% RSLogix 500 project Project_2.RSS, saved by version 8.30.00.16 %
PROJECT "UNTITLED"    % processor: Bul.1763 MicroLogix 1100 Series A %

PROGRAM FILES
  LAD 2   3 rungs
  LAD 3 "IO"  8 rungs  % Digital IO %
  LAD 4 "LOGIC"  12 rungs

DATA FILES
  O0 OUTPUT  4 elements
  I1 INPUT  6 elements
  S2 STATUS  66 elements
  B3 BINARY  1 elements
  T4 TIMER  4 elements
  C5 COUNTER  1 elements
  R6 CONTROL  1 elements
  N7 INTEGER  1 elements
  F8 FLOAT  1 elements

LADDER 2
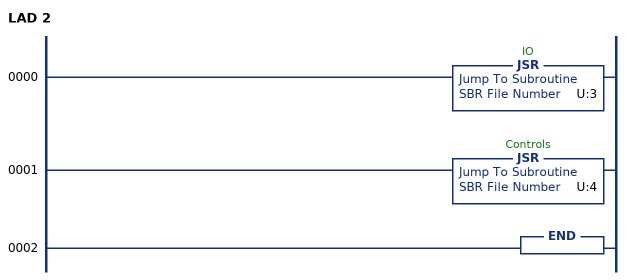
% Rung: 0 %
SOR JSR U:3 EOR
%   U:3  "IO" %
% Rung: 1 %
SOR JSR U:4 EOR
%   U:4  "Controls" %
% Rung: 2 %
SOR END EOR

LADDER 3 "IO"    % Digital IO %
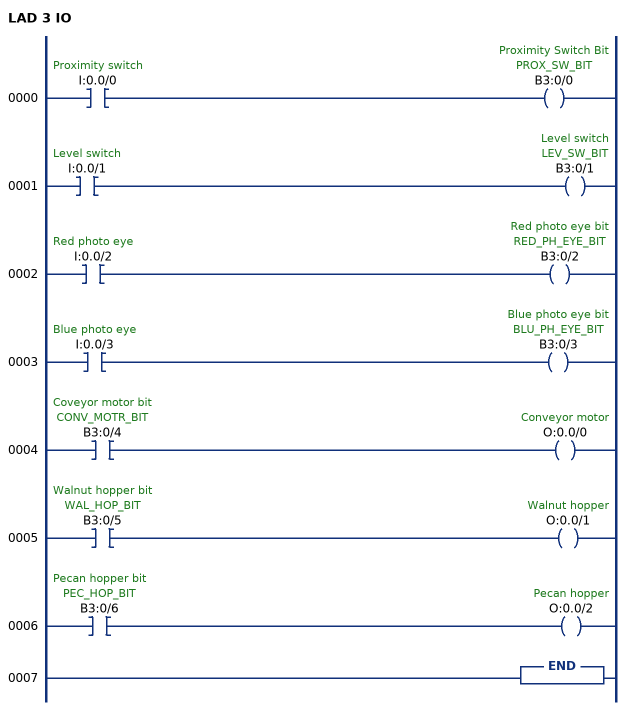
% Rung: 0 %
SOR XIC I:0.0/0 OTE B3:0/0 EOR
%   I:0.0/0  "Proximity switch" %
%   B3:0/0  PROX_SW_BIT  "Proximity Switch Bit" %
% Rung: 1 %
SOR XIC I:0.0/1 OTE B3:0/1 EOR
%   I:0.0/1  "Level switch" %
%   B3:0/1  LEV_SW_BIT  "Level switch" %
% Rung: 2 %
SOR XIC I:0.0/2 OTE B3:0/2 EOR
%   I:0.0/2  "Red photo eye" %
%   B3:0/2  RED_PH_EYE_BIT  "Red photo eye bit" %
% Rung: 3 %
SOR XIC I:0.0/3 OTE B3:0/3 EOR
%   I:0.0/3  "Blue photo eye" %
%   B3:0/3  BLU_PH_EYE_BIT  "Blue photo eye bit" %
% Rung: 4 %
SOR XIC B3:0/4 OTE O:0.0/0 EOR
%   B3:0/4  CONV_MOTR_BIT  "Coveyor motor bit" %
%   O:0.0/0  "Conveyor motor" %
% Rung: 5 %
SOR XIC B3:0/5 OTE O:0.0/1 EOR
%   B3:0/5  WAL_HOP_BIT  "Walnut hopper bit" %
%   O:0.0/1  "Walnut hopper" %
% Rung: 6 %
SOR XIC B3:0/6 OTE O:0.0/2 EOR
%   B3:0/6  PEC_HOP_BIT  "Pecan hopper bit" %
%   O:0.0/2  "Pecan hopper" %
% Rung: 7 %
SOR END EOR

LADDER 4 "LOGIC"
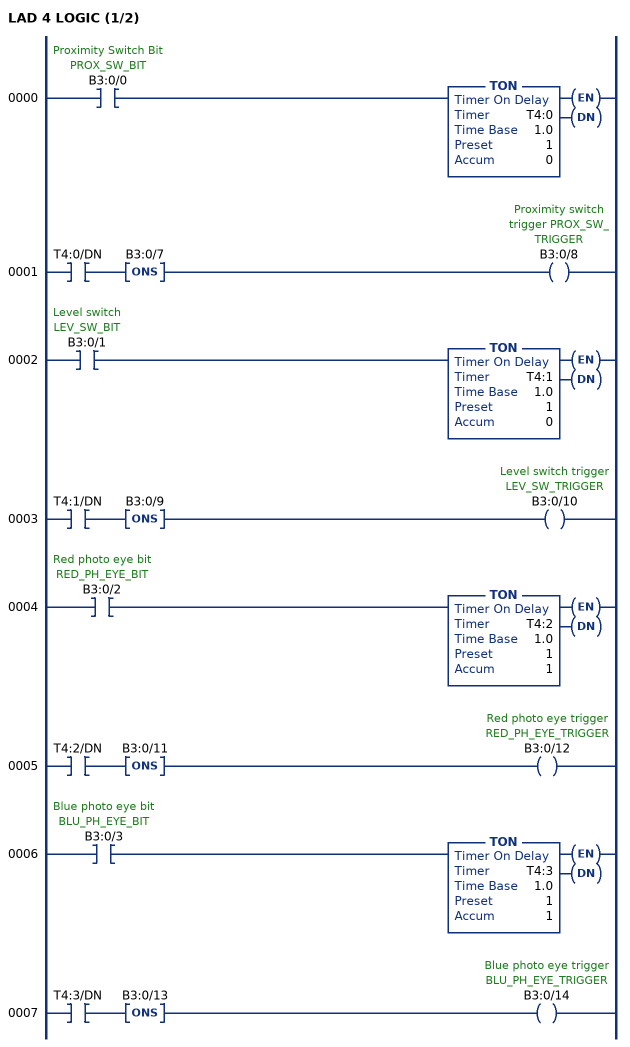
% Rung: 0 %
SOR XIC B3:0/0 TON T4:0 1.0 1 0 EOR
%   B3:0/0  PROX_SW_BIT  "Proximity Switch Bit" %
% Rung: 1 %
SOR XIC T4:0/DN ONS B3:0/7 OTE B3:0/8 EOR
%   B3:0/8  PROX_SW_TRIGGER  "Proximity switch trigger" %
% Rung: 2 %
SOR XIC B3:0/1 TON T4:1 1.0 1 0 EOR
%   B3:0/1  LEV_SW_BIT  "Level switch" %
% Rung: 3 %
SOR XIC T4:1/DN ONS B3:0/9 OTE B3:0/10 EOR
%   B3:0/10  LEV_SW_TRIGGER  "Level switch trigger" %
% Rung: 4 %
SOR XIC B3:0/2 TON T4:2 1.0 1 1 EOR
%   B3:0/2  RED_PH_EYE_BIT  "Red photo eye bit" %
% Rung: 5 %
SOR XIC T4:2/DN ONS B3:0/11 OTE B3:0/12 EOR
%   B3:0/12  RED_PH_EYE_TRIGGER  "Red photo eye trigger" %
% Rung: 6 %
SOR XIC B3:0/3 TON T4:3 1.0 1 1 EOR
%   B3:0/3  BLU_PH_EYE_BIT  "Blue photo eye bit" %
% Rung: 7 %
SOR XIC T4:3/DN ONS B3:0/13 OTE B3:0/14 EOR
%   B3:0/14  BLU_PH_EYE_TRIGGER  "Blue photo eye trigger" %

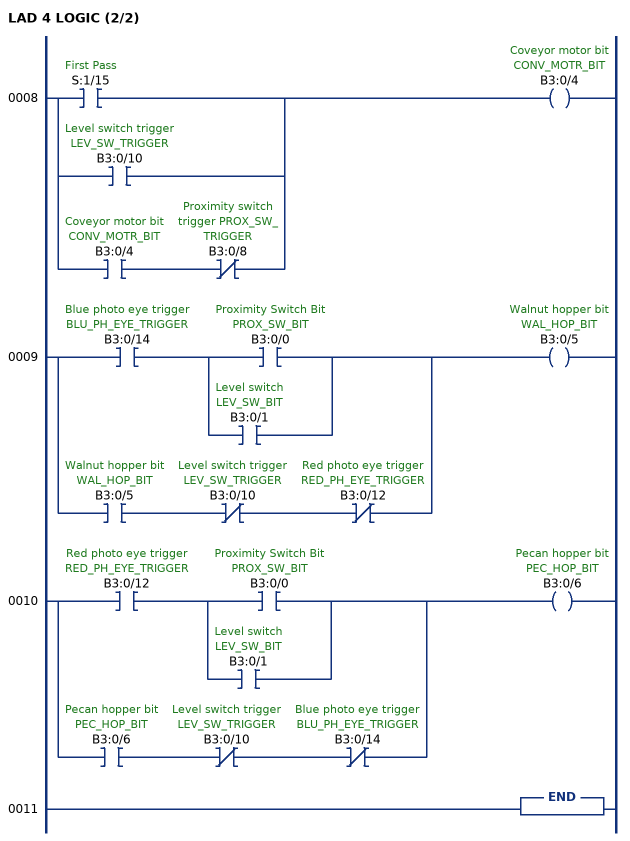
% Rung: 8 %
SOR BST BST XIC S:1/15 NXB XIC B3:0/10 BND NXB XIC B3:0/4 XIO B3:0/8 BND OTE B3:0/4 EOR
%   S:1/15  "First Pass" %
%   B3:0/10  LEV_SW_TRIGGER  "Level switch trigger" %
%   B3:0/4  CONV_MOTR_BIT  "Coveyor motor bit" %
%   B3:0/8  PROX_SW_TRIGGER  "Proximity switch trigger" %
% Rung: 9 %
SOR BST XIC B3:0/14 BST XIC B3:0/0 NXB XIC B3:0/1 BND NXB XIC B3:0/5 XIO B3:0/10 XIO B3:0/12 BND OTE B3:0/5 EOR
%   B3:0/14  BLU_PH_EYE_TRIGGER  "Blue photo eye trigger" %
%   B3:0/0  PROX_SW_BIT  "Proximity Switch Bit" %
%   B3:0/1  LEV_SW_BIT  "Level switch" %
%   B3:0/5  WAL_HOP_BIT  "Walnut hopper bit" %
%   B3:0/10  LEV_SW_TRIGGER  "Level switch trigger" %
%   B3:0/12  RED_PH_EYE_TRIGGER  "Red photo eye trigger" %
% Rung: 10 %
SOR BST XIC B3:0/12 BST XIC B3:0/0 NXB XIC B3:0/1 BND NXB XIC B3:0/6 XIO B3:0/10 XIO B3:0/14 BND OTE B3:0/6 EOR
%   B3:0/12  RED_PH_EYE_TRIGGER  "Red photo eye trigger" %
%   B3:0/0  PROX_SW_BIT  "Proximity Switch Bit" %
%   B3:0/1  LEV_SW_BIT  "Level switch" %
%   B3:0/6  PEC_HOP_BIT  "Pecan hopper bit" %
%   B3:0/10  LEV_SW_TRIGGER  "Level switch trigger" %
%   B3:0/14  BLU_PH_EYE_TRIGGER  "Blue photo eye trigger" %
% Rung: 11 %
SOR END EOR

DATA TABLE (non-zero values as saved)
DATA B3
% B3:0 % 0X281C
DATA T4
% .PRE .ACC %
% T4:0 % 1 0
% T4:1 % 1 0
% T4:2 % 1 1
% T4:3 % 1 1
